// TIA Portal V17 export
// export: Created 2024-09-15T12:30:30.5077414Z, ExportSetting WithDefaults, DisplayName Totally Integrated Automation Portal, DisplayVersion V17, DisplayName TIA Portal Openness, DisplayVersion V17, DisplayName TIA Portal Version Control Interface, DisplayVersion V17, DisplayName STEP 7 Professional, DisplayVersion V17, DisplayName STEP 7 Safety, DisplayVersion V17, DisplayName WinCC Professional, DisplayVersion V17
TYPE "typ_HBW"
// stored: IsFailsafeCompliant false
   STRUCT
      x_Start_Park_Position : Bool;
      x_Park_Position_Reached : Bool;
      x_HBW_PickedUp_Accepted : Bool;
      x_HBW_Discards_Accepted : Bool;
      x_HBW_PickUp_Ready : Bool;
      x_HBW_Container_Available : Bool;
      x_Error : Bool;
      s_ErrorMessage : String;
      di_PosBelt_Horizontal : DInt;
      di_PosBelt_Vertical : DInt;
      di_Offset_Pos_Belt_Vertical : DInt;
      di_PosRack_A1_Horizontal : DInt;
      di_PosRack_A1_Vertical : DInt;
      di_PosRack_B2_Horizontal : DInt;
      di_PosRack_B2_Vertical : DInt;
      di_PosRack_C3_Horizontal : DInt;
      di_PosRack_C3_Vertical : DInt;
      di_Offset_Pos_Rack_Vertical : DInt;
      di_Pos_Park_Horizontal : DInt;
      di_Pos_Park_Vertical : DInt;
      i_PWM_ConveyorBelt : Int := 800;
      i_PWM_Cantilever : Int := 800;
      Workpiece : "typ_Workpiece";
      History : Array[1..20] of "typ_History";
      Rack_Pos : Array[1..3, 1..3] of "typ_Rack_Pos";
      Rack_Workpiece : Array[1..3, 1..3] of "typ_Workpiece";
      Rack_History : Array[1..3, 1..3] of "typ_Rack_History";
      Horizontal_Axis : "typ_Axis";
      Vertical_Axis : "typ_Axis";
      i_Red_Available { S7_SetPoint := 'True'} : Int;
      i_Blue_Available : Int;
      i_White_Available : Int;
      di_Offset_Actual_Pickup : DInt;
   END_STRUCT;
END_TYPE
